// TIA Portal V19 export
TYPE "LAF_typeAxisDiagStatusPositioning"
TITLE = LAF_typeAxisDiagStatusPositioning
// Status information about a positioning motion of a Technology Object
// stored: Access Published
   STRUCT
      targetPosition { ExternalWritable := 'False'} : LReal;   // Target position
      followingError { ExternalWritable := 'False'} : LReal;   // Current following error
   END_STRUCT;
END_TYPE
